ABB RAPID module: 0069C0E9

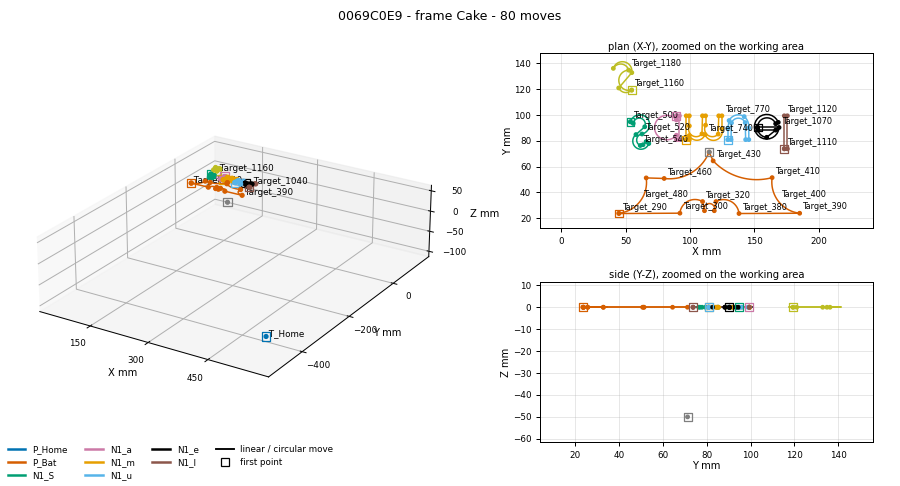
[picture p0: tool path of 0069C0E9 in frame Cake, 80 of 80 moves have a stored position in this frame; points joined in program order, loops and branches not executed]
MODULE Module1
    CONST robtarget T_Home:=[[572.610973065,-505,-40.400436373],[0,-0.000000007,0,1],[0,0,0,0],[9E+09,9E+09,9E+09,9E+09,9E+09,9E+09]];
    CONST robtarget Target_10:=[[44.887,23.575,0],[0.707106781,0,0,-0.707106781],[0,0,0,0],[9E+09,9E+09,9E+09,9E+09,9E+09,9E+09]];
    CONST robtarget Target_20:=[[91.921,23.575,0],[0.707106781,0,0,-0.707106781],[0,0,0,0],[9E+09,9E+09,9E+09,9E+09,9E+09,9E+09]];
    CONST robtarget Target_30:=[[93.942,29.137,0],[0.707106781,0,0,-0.707106781],[0,0,0,0],[9E+09,9E+09,9E+09,9E+09,9E+09,9E+09]];
    CONST robtarget Target_40:=[[97.861,32.778,0],[0.707106781,0,0,-0.707106781],[0,0,0,0],[9E+09,9E+09,9E+09,9E+09,9E+09,9E+09]];
    CONST robtarget Target_50:=[[101.269,33.587,0],[0.707106781,0,0,-0.707106781],[0,0,0,0],[9E+09,9E+09,9E+09,9E+09,9E+09,9E+09]];
    CONST robtarget Target_60:=[[104.374,34.284,0],[0.707106781,0,0,-0.707106781],[0,0,0,0],[9E+09,9E+09,9E+09,9E+09,9E+09,9E+09]];
    CONST robtarget Target_70:=[[107.601,34.604,0],[0.707106781,0,0,-0.707106781],[0,0,0,0],[9E+09,9E+09,9E+09,9E+09,9E+09,9E+09]];
    CONST robtarget Target_80:=[[109.794,32.852,0],[0.707106781,0,0,-0.707106781],[0,0,0,0],[9E+09,9E+09,9E+09,9E+09,9E+09,9E+09]];
    CONST robtarget Target_90:=[[111.194,25.675,0],[0.707106781,0,0,-0.707106781],[0,0,0,0],[9E+09,9E+09,9E+09,9E+09,9E+09,9E+09]];
    CONST robtarget Target_100:=[[112.426,30.409,0],[0.707106781,0,0,-0.707106781],[0,0,0,0],[9E+09,9E+09,9E+09,9E+09,9E+09,9E+09]];
    CONST robtarget Target_110:=[[115,30.175,0],[0.707106781,0,0,-0.707106781],[0,0,0,0],[9E+09,9E+09,9E+09,9E+09,9E+09,9E+09]];
    CONST robtarget Target_120:=[[117.574,30.409,0],[0.707106781,0,0,-0.707106781],[0,0,0,0],[9E+09,9E+09,9E+09,9E+09,9E+09,9E+09]];
    CONST robtarget Target_130:=[[118.806,25.675,0],[0.707106781,0,0,-0.707106781],[0,0,0,0],[9E+09,9E+09,9E+09,9E+09,9E+09,9E+09]];
    CONST robtarget Target_140:=[[120.206,32.852,0],[0.707106781,0,0,-0.707106781],[0,0,0,0],[9E+09,9E+09,9E+09,9E+09,9E+09,9E+09]];
    CONST robtarget Target_150:=[[122.399,34.604,0],[0.707106781,0,0,-0.707106781],[0,0,0,0],[9E+09,9E+09,9E+09,9E+09,9E+09,9E+09]];
    CONST robtarget Target_160:=[[125.626,34.284,0],[0.707106781,0,0,-0.707106781],[0,0,0,0],[9E+09,9E+09,9E+09,9E+09,9E+09,9E+09]];
    CONST robtarget Target_170:=[[128.731,33.587,0],[0.707106781,0,0,-0.707106781],[0,0,0,0],[9E+09,9E+09,9E+09,9E+09,9E+09,9E+09]];
    CONST robtarget Target_180:=[[132.139,32.778,0],[0.707106781,0,0,-0.707106781],[0,0,0,0],[9E+09,9E+09,9E+09,9E+09,9E+09,9E+09]];
    CONST robtarget Target_190:=[[136.058,29.137,0],[0.707106781,0,0,-0.707106781],[0,0,0,0],[9E+09,9E+09,9E+09,9E+09,9E+09,9E+09]];
    CONST robtarget Target_200:=[[137.882,23.65,0],[0.707106781,0,0,-0.707106781],[0,0,0,0],[9E+09,9E+09,9E+09,9E+09,9E+09,9E+09]];
    CONST robtarget Target_210:=[[185.214,23.669,0],[0.707106781,0,0,-0.707106781],[0,0,0,0],[9E+09,9E+09,9E+09,9E+09,9E+09,9E+09]];
    CONST robtarget Target_220:=[[168.341,33.479,0],[0.707106781,0,0,-0.707106781],[0,0,0,0],[9E+09,9E+09,9E+09,9E+09,9E+09,9E+09]];
    CONST robtarget Target_230:=[[163.916,51.359,0],[0.707106781,0,0,-0.707106781],[0,0,0,0],[9E+09,9E+09,9E+09,9E+09,9E+09,9E+09]];
    CONST robtarget Target_240:=[[135.263,52.898,0],[0.707106781,0,0,-0.707106781],[0,0,0,0],[9E+09,9E+09,9E+09,9E+09,9E+09,9E+09]];
    CONST robtarget Target_250:=[[114.922,71.263,0],[0.707106781,0,0,-0.707106781],[0,0,0,0],[9E+09,9E+09,9E+09,9E+09,9E+09,9E+09]];
    CONST robtarget Target_260:=[[94.738,52.898,0],[0.707106781,0,0,-0.707106781],[0,0,0,0],[9E+09,9E+09,9E+09,9E+09,9E+09,9E+09]];
    CONST robtarget Target_270:=[[66.084,51.359,0],[0.707106781,0,0,-0.707106781],[0,0,0,0],[9E+09,9E+09,9E+09,9E+09,9E+09,9E+09]];
    CONST robtarget Target_280:=[[61.659,33.479,0],[0.707106781,0,0,-0.707106781],[0,0,0,0],[9E+09,9E+09,9E+09,9E+09,9E+09,9E+09]];
    CONST robtarget Target_290:=[[44.887375283,23.575,0],[0.707106781,0,0,-0.707106781],[0,0,0,0],[9E+09,9E+09,9E+09,9E+09,9E+09,9E+09]];
    CONST robtarget Target_300:=[[92.217626762,23.834877014,0],[0.5,0,0,-0.866025404],[-1,0,-1,0],[9E+09,9E+09,9E+09,9E+09,9E+09,9E+09]];
    CONST robtarget Target_400:=[[168.340891695,33.478608179,0],[0.5,0,0,-0.866025404],[-1,0,-1,0],[9E+09,9E+09,9E+09,9E+09,9E+09,9E+09]];
    CONST robtarget Target_430:=[[118.021503486,64.425747652,0],[0.5,0,0,-0.866025404],[0,0,0,0],[9E+09,9E+09,9E+09,9E+09,9E+09,9E+09]];
    CONST robtarget Target_310:=[[97.860623741,32.777873993,0],[0.5,0,0,-0.866025404],[-1,0,-1,0],[9E+09,9E+09,9E+09,9E+09,9E+09,9E+09]];
    CONST robtarget Target_480:=[[61.659109682,33.478608179,0],[0.5,0,0,-0.866025404],[-1,0,-1,0],[9E+09,9E+09,9E+09,9E+09,9E+09,9E+09]];
    CONST robtarget Target_420:=[[135.262514114,52.897562122,0],[0.5,0,0,-0.866025404],[-1,0,-1,0],[9E+09,9E+09,9E+09,9E+09,9E+09,9E+09]];
    CONST robtarget Target_460:=[[79.985840188,50.770867258,0],[0.5,0,0,-0.866025404],[0,0,0,0],[9E+09,9E+09,9E+09,9E+09,9E+09,9E+09]];
    CONST robtarget Target_330:=[[111.283377266,25.744747734,0],[0.5,0,0,-0.866025404],[-1,0,-1,0],[9E+09,9E+09,9E+09,9E+09,9E+09,9E+09]];
    CONST robtarget Target_380:=[[138.079373741,23.575,0],[0.5,0,0,-0.866025404],[0,0,0,0],[9E+09,9E+09,9E+09,9E+09,9E+09,9E+09]];
    CONST robtarget Target_340:=[[112.525,30.426625252,0],[0.5,0,0,-0.866025404],[-1,0,-1,0],[9E+09,9E+09,9E+09,9E+09,9E+09,9E+09]];
    CONST robtarget Target_490:=[[44.854375315,23.789501762,0],[0.707106781,0,0,-0.707106781],[0,0,0,0],[9E+09,9E+09,9E+09,9E+09,9E+09,9E+09]];
    CONST robtarget Target_360:=[[120.205747986,32.852127266,0],[0.5,0,0,-0.866025404],[-1,0,-1,0],[9E+09,9E+09,9E+09,9E+09,9E+09,9E+09]];
    CONST robtarget Target_350:=[[118.898123741,25.740625,0],[0.5,0,0,-0.866025404],[0,0,0,0],[9E+09,9E+09,9E+09,9E+09,9E+09,9E+09]];
    CONST robtarget Target_370:=[[132.139376259,32.777873993,0],[0.5,0,0,-0.866025404],[-1,0,-1,0],[9E+09,9E+09,9E+09,9E+09,9E+09,9E+09]];
    CONST robtarget Target_410:=[[163.773995972,51.414627266,0],[0.5,0,0,-0.866025404],[0,0,0,0],[9E+09,9E+09,9E+09,9E+09,9E+09,9E+09]];
    CONST robtarget Target_470:=[[66.061000252,51.208377266,0],[0.5,0,0,-0.866025404],[-1,0,-1,0],[9E+09,9E+09,9E+09,9E+09,9E+09,9E+09]];
    CONST robtarget Target_320:=[[109.794252014,32.852127266,0],[0.5,0,0,-0.866025404],[0,0,0,0],[9E+09,9E+09,9E+09,9E+09,9E+09,9E+09]];
    CONST robtarget Target_440:=[[114.884500504,71.210504532,0],[0.5,0,0,-0.866025404],[-1,0,-1,0],[9E+09,9E+09,9E+09,9E+09,9E+09,9E+09]];
    CONST robtarget Target_450:=[[101.522546531,55.448907324,0],[0.5,0,0,-0.866025404],[-1,0,-1,0],[9E+09,9E+09,9E+09,9E+09,9E+09,9E+09]];
    CONST robtarget Target_390:=[[185.145619965,23.789501762,0],[0.5,0,0,-0.866025404],[-1,0,-1,0],[9E+09,9E+09,9E+09,9E+09,9E+09,9E+09]];
    CONST robtarget Target_500:=[[53.851116523,94.745073318,0],[0.707106781,0,0,-0.707106781],[0,0,0,0],[9E+09,9E+09,9E+09,9E+09,9E+09,9E+09]];
    CONST robtarget Target_510:=[[66.419099197,98.025150299,0],[0.707106781,0,0,-0.707106781],[-1,-1,0,0],[9E+09,9E+09,9E+09,9E+09,9E+09,9E+09]];
    CONST robtarget Target_520:=[[62.824605331,85.278720856,0],[0.707106781,0,0,-0.707106781],[0,0,0,0],[9E+09,9E+09,9E+09,9E+09,9E+09,9E+09]];
    CONST robtarget Target_530:=[[58.834970817,81.913661957,0],[0.707106781,0,0,-0.707106781],[-1,-1,0,0],[9E+09,9E+09,9E+09,9E+09,9E+09,9E+09]];
    CONST robtarget Target_540:=[[61.44799076,76.356220245,0],[0.707106781,0,0,-0.707106781],[0,0,0,0],[9E+09,9E+09,9E+09,9E+09,9E+09,9E+09]];
    CONST robtarget Target_550:=[[63.614881858,76.951055527,0],[0.707106781,0,0,-0.707106781],[-1,-1,0,0],[9E+09,9E+09,9E+09,9E+09,9E+09,9E+09]];
    CONST robtarget Target_560:=[[66.01970993,79.415369034,0],[0.707106781,0,0,-0.707106781],[-1,-1,0,0],[9E+09,9E+09,9E+09,9E+09,9E+09,9E+09]];
    CONST robtarget Target_570:=[[68.059137687,77.868800163,0],[0.707106781,0,0,-0.707106781],[-1,-1,0,0],[9E+09,9E+09,9E+09,9E+09,9E+09,9E+09]];
    CONST robtarget Target_580:=[[58.414338455,74.546232224,0],[0.707106781,0,0,-0.707106781],[-1,-1,0,0],[9E+09,9E+09,9E+09,9E+09,9E+09,9E+09]];
    CONST robtarget Target_590:=[[58.112676963,84.841098785,0],[0.707106781,0,0,-0.707106781],[0,0,0,0],[9E+09,9E+09,9E+09,9E+09,9E+09,9E+09]];
    CONST robtarget Target_600:=[[64.932015762,90.887155533,0],[0.707106781,0,0,-0.707106781],[-1,-1,0,0],[9E+09,9E+09,9E+09,9E+09,9E+09,9E+09]];
    CONST robtarget Target_610:=[[61.159070358,97.600269318,0],[0.707106781,0,0,-0.707106781],[-1,-1,0,0],[9E+09,9E+09,9E+09,9E+09,9E+09,9E+09]];
    CONST robtarget Target_620:=[[55.97552143,93.470430374,0],[0.707106781,0,0,-0.707106781],[0,0,0,0],[9E+09,9E+09,9E+09,9E+09,9E+09,9E+09]];
    CONST robtarget Target_630:=[[89.456146583,99.401769638,0],[0.608761429,0,0,-0.79335334],[0,0,0,0],[9E+09,9E+09,9E+09,9E+09,9E+09,9E+09]];
    CONST robtarget Target_640:=[[91.801489219,99.401769638,0],[0.608761429,0,0,-0.79335334],[-1,0,-1,0],[9E+09,9E+09,9E+09,9E+09,9E+09,9E+09]];
    CONST robtarget Target_650:=[[91.801489219,80.910949707,0],[0.608761429,0,0,-0.79335334],[-1,0,-1,0],[9E+09,9E+09,9E+09,9E+09,9E+09,9E+09]];
    CONST robtarget Target_660:=[[89.456146583,80.910949707,0],[0.608761429,0,0,-0.79335334],[-1,0,-1,0],[9E+09,9E+09,9E+09,9E+09,9E+09,9E+09]];
    CONST robtarget Target_670:=[[89.456146583,84.309997559,0],[0.608761429,0,0,-0.79335334],[-1,0,-1,0],[9E+09,9E+09,9E+09,9E+09,9E+09,9E+09]];
    CONST robtarget Target_680:=[[72.545884475,90.105371475,0],[0.608761429,0,0,-0.79335334],[-1,0,-1,0],[9E+09,9E+09,9E+09,9E+09,9E+09,9E+09]];
    CONST robtarget Target_690:=[[89.456146583,96.223659515,0],[0.608761429,0,0,-0.79335334],[0,0,0,0],[9E+09,9E+09,9E+09,9E+09,9E+09,9E+09]];
    CONST robtarget Target_700:=[[97.138002738,80.910949707,0],[0.608761429,0,0,-0.793353341],[0,0,0,0],[9E+09,9E+09,9E+09,9E+09,9E+09,9E+09]];
    CONST robtarget Target_710:=[[99.51732479,80.910949707,0],[0.608761429,0,0,-0.793353341],[-1,0,-1,0],[9E+09,9E+09,9E+09,9E+09,9E+09,9E+09]];
    CONST robtarget Target_720:=[[99.51732479,84.106054306,0],[0.608761429,0,0,-0.793353341],[-1,0,-1,0],[9E+09,9E+09,9E+09,9E+09,9E+09,9E+09]];
    CONST robtarget Target_730:=[[105.863989219,80.435085297,0],[0.608761429,0,0,-0.793353341],[-1,0,-1,0],[9E+09,9E+09,9E+09,9E+09,9E+09,9E+09]];
    CONST robtarget Target_740:=[[111.716993675,84.870834351,0],[0.608761429,0,0,-0.793353341],[0,0,0,0],[9E+09,9E+09,9E+09,9E+09,9E+09,9E+09]];
    CONST robtarget Target_750:=[[121.89846836,81.403808594,0],[0.608761429,0,0,-0.793353341],[-1,0,-1,0],[9E+09,9E+09,9E+09,9E+09,9E+09,9E+09]];
    CONST robtarget Target_760:=[[124.789255485,89.306592941,0],[0.608761429,0,0,-0.793353341],[0,0,0,0],[9E+09,9E+09,9E+09,9E+09,9E+09,9E+09]];
    CONST robtarget Target_770:=[[124.789255485,99.401769638,0],[0.608761429,0,0,-0.793353341],[-1,0,-1,0],[9E+09,9E+09,9E+09,9E+09,9E+09,9E+09]];
    CONST robtarget Target_780:=[[122.35893093,99.401769638,0],[0.608761429,0,0,-0.793353341],[-1,0,-1,0],[9E+09,9E+09,9E+09,9E+09,9E+09,9E+09]];
    CONST robtarget Target_790:=[[121.935518607,85.219240189,0],[0.608761429,0,0,-0.793353341],[-1,0,-1,0],[9E+09,9E+09,9E+09,9E+09,9E+09,9E+09]];
    CONST robtarget Target_800:=[[114.880369529,83.766145706,0],[0.608761429,0,0,-0.793353341],[-1,0,-1,0],[9E+09,9E+09,9E+09,9E+09,9E+09,9E+09]];
    CONST robtarget Target_810:=[[112.127798423,92.161798477,0],[0.608761429,0,0,-0.793353341],[0,0,0,0],[9E+09,9E+09,9E+09,9E+09,9E+09,9E+09]];
    CONST robtarget Target_820:=[[112.127798423,99.401769638,0],[0.608761429,0,0,-0.793353341],[-1,0,-1,0],[9E+09,9E+09,9E+09,9E+09,9E+09,9E+09]];
    CONST robtarget Target_830:=[[109.748466834,99.401769638,0],[0.608761429,0,0,-0.793353341],[-1,0,-1,0],[9E+09,9E+09,9E+09,9E+09,9E+09,9E+09]];
    CONST robtarget Target_840:=[[109.332083091,85.389194489,0],[0.608761429,0,0,-0.793353341],[-1,0,-1,0],[9E+09,9E+09,9E+09,9E+09,9E+09,9E+09]];
    CONST robtarget Target_850:=[[102.330044135,83.740653992,0],[0.608761429,0,0,-0.793353341],[-1,0,-1,0],[9E+09,9E+09,9E+09,9E+09,9E+09,9E+09]];
    CONST robtarget Target_860:=[[99.51732479,91.566963196,0],[0.608761429,0,0,-0.793353341],[0,0,0,0],[9E+09,9E+09,9E+09,9E+09,9E+09,9E+09]];
    CONST robtarget Target_870:=[[99.51732479,99.401769638,0],[0.608761429,0,0,-0.793353341],[-1,0,-1,0],[9E+09,9E+09,9E+09,9E+09,9E+09,9E+09]];
    CONST robtarget Target_880:=[[97.138002738,99.401769638,0],[0.608761429,0,0,-0.793353341],[-1,0,-1,0],[9E+09,9E+09,9E+09,9E+09,9E+09,9E+09]];
    CONST robtarget Target_890:=[[129.496935233,80.910949707,0],[0.5,0,0,-0.866025404],[0,0,0,0],[9E+09,9E+09,9E+09,9E+09,9E+09,9E+09]];
    CONST robtarget Target_900:=[[131.876266822,80.910949707,0],[0.5,0,0,-0.866025404],[-1,0,-1,0],[9E+09,9E+09,9E+09,9E+09,9E+09,9E+09]];
    CONST robtarget Target_910:=[[132.216699943,93.895311356,0],[0.5,0,0,-0.866025404],[-1,0,-1,0],[9E+09,9E+09,9E+09,9E+09,9E+09,9E+09]];
    CONST robtarget Target_920:=[[137.595165595,97.566280365,0],[0.5,0,0,-0.866025404],[-1,0,-1,0],[9E+09,9E+09,9E+09,9E+09,9E+09,9E+09]];
    CONST robtarget Target_930:=[[142.88864933,94.082260132,0],[0.5,0,0,-0.866025404],[0,0,0,0],[9E+09,9E+09,9E+09,9E+09,9E+09,9E+09]];
    CONST robtarget Target_940:=[[143.246086463,80.910949707,0],[0.5,0,0,-0.866025404],[-1,0,-1,0],[9E+09,9E+09,9E+09,9E+09,9E+09,9E+09]];
    CONST robtarget Target_950:=[[145.676401481,80.910949707,0],[0.5,0,0,-0.866025404],[-1,0,-1,0],[9E+09,9E+09,9E+09,9E+09,9E+09,9E+09]];
    CONST robtarget Target_1000:=[[145.676,89.986,0],[0.5,0,0,-0.866025404],[-1,0,-1,0],[9E+09,9E+09,9E+09,9E+09,9E+09,9E+09]];
    CONST robtarget Target_960:=[[145.453346595,93.338718414,0],[0.5,0,0,-0.866025404],[-1,0,-1,0],[9E+09,9E+09,9E+09,9E+09,9E+09,9E+09]];
    CONST robtarget Target_970:=[[142.098911628,98.781442642,0],[0.5,0,0,-0.866025404],[-1,0,-1,0],[9E+09,9E+09,9E+09,9E+09,9E+09,9E+09]];
    CONST robtarget Target_980:=[[133.091429099,98.781442642,0],[0.5,0,0,-0.866025404],[-1,0,-1,0],[9E+09,9E+09,9E+09,9E+09,9E+09,9E+09]];
    CONST robtarget Target_1010:=[[130.389,95.722,0],[0.5,0,0,-0.866025404],[-1,0,-1,0],[9E+09,9E+09,9E+09,9E+09,9E+09,9E+09]];
    CONST robtarget Target_990:=[[129.496935233,89.816455841,0],[0.5,0,0,-0.866025404],[0,0,0,0],[9E+09,9E+09,9E+09,9E+09,9E+09,9E+09]];
    CONST robtarget Target_1020:=[[152.508495674,90.34330368,0],[0.5,0,0,-0.866025404],[0,0,0,0],[9E+09,9E+09,9E+09,9E+09,9E+09,9E+09]];
    CONST robtarget Target_1030:=[[156.792162284,97.170209885,0],[0.5,0,0,-0.866025404],[-1,0,-1,0],[9E+09,9E+09,9E+09,9E+09,9E+09,9E+09]];
    CONST robtarget Target_1040:=[[166.529577598,93.266487122,0],[0.5,0,0,-0.866025404],[0,0,0,0],[9E+09,9E+09,9E+09,9E+09,9E+09,9E+09]];
    CONST robtarget Target_1050:=[[168.535002097,94.320192337,0],[0.5,0,0,-0.866025404],[-1,0,-1,0],[9E+09,9E+09,9E+09,9E+09,9E+09,9E+09]];
    CONST robtarget Target_1060:=[[150.061176643,90.20734787,0],[0.5,0,0,-0.866025404],[-1,0,-1,0],[9E+09,9E+09,9E+09,9E+09,9E+09,9E+09]];
    CONST robtarget Target_1070:=[[169.146841392,90.34330368,0],[0.5,0,0,-0.866025404],[0,0,0,0],[9E+09,9E+09,9E+09,9E+09,9E+09,9E+09]];
    CONST robtarget Target_1020_2:=[[152.508495674,90.34330368,0],[0.5,0,0,-0.866025404],[0,0,0,0],[9E+09,9E+09,9E+09,9E+09,9E+09,9E+09]];
    CONST robtarget Target_1080:=[[152.746,88.287,0],[0.5,0,0,-0.866025404],[-1,0,-1,0],[9E+09,9E+09,9E+09,9E+09,9E+09,9E+09]];
    CONST robtarget Target_1090:=[[159.587,82.712,0],[0.5,0,0,-0.866025404],[-1,0,-1,0],[9E+09,9E+09,9E+09,9E+09,9E+09,9E+09]];
    CONST robtarget Target_1100:=[[166.53,88.287,0],[0.5,0,0,-0.866025404],[-1,0,-1,0],[9E+09,9E+09,9E+09,9E+09,9E+09,9E+09]];
    CONST robtarget Target_1110:=[[173.225706443,73.772945404,0],[0.5,0,0,-0.866025404],[0,0,0,0],[9E+09,9E+09,9E+09,9E+09,9E+09,9E+09]];
    CONST robtarget Target_1120:=[[173.225706443,99.401769638,0],[0.5,0,0,-0.866025404],[-1,0,-1,0],[9E+09,9E+09,9E+09,9E+09,9E+09,9E+09]];
    CONST robtarget Target_1130:=[[175.605028495,99.401769638,0],[0.5,0,0,-0.866025404],[-1,0,-1,0],[9E+09,9E+09,9E+09,9E+09,9E+09,9E+09]];
    CONST robtarget Target_1140:=[[175.605028495,73.772945404,0],[0.5,0,0,-0.866025404],[-1,0,-1,0],[9E+09,9E+09,9E+09,9E+09,9E+09,9E+09]];
    CONST robtarget Target_1150:=[[173.225706443,73.772945404,0],[0.5,0,0,-0.866025404],[-1,0,-1,0],[9E+09,9E+09,9E+09,9E+09,9E+09,9E+09]];
    CONST robtarget T_Local_Home:=[[115.079,71.263,-50],[0.707106781,0.000000005,-0.000000005,-0.707106781],[0,0,0,0],[9E+09,9E+09,9E+09,9E+09,9E+09,9E+09]];

    ! Variable para almacenar posición temporal
    VAR robtarget current_pos;
    CONST robtarget Target_1160:=[[54.76886116,119.337177277,0],[0.446392083,0,0,-0.894837476],[0,0,0,0],[9E+09,9E+09,9E+09,9E+09,9E+09,9E+09]];
    CONST robtarget Target_1170:=[[44.822400436,126.309480667,0],[0.36650971,0,0,-0.930414226],[0,0,0,0],[9E+09,9E+09,9E+09,9E+09,9E+09,9E+09]];
    CONST robtarget Target_1180:=[[52.491501197,134.819850922,0],[0.740357165,0,0,0.672213707],[0,0,0,0],[9E+09,9E+09,9E+09,9E+09,9E+09,9E+09]];
    CONST robtarget Target_1190:=[[49.088199958,138.922071457,0],[0.121523417,0,0,0.992588565],[0,0,0,0],[9E+09,9E+09,9E+09,9E+09,9E+09,9E+09]];
    CONST robtarget Target_1200:=[[40.560839996,136.2134552,0],[0.266933582,0,0,0.963714928],[0,0,0,0],[9E+09,9E+09,9E+09,9E+09,9E+09,9E+09]];
    CONST robtarget Target_1210:=[[45.935591087,141.1951828,0],[0.989624414,0,0,0.143678526],[0,0,0,0],[9E+09,9E+09,9E+09,9E+09,9E+09,9E+09]];
    CONST robtarget Target_1220:=[[54.89208065,132.886638641,0],[0.594295659,0,0,-0.804246648],[0,0,0,0],[9E+09,9E+09,9E+09,9E+09,9E+09,9E+09]];
    CONST robtarget Target_1230:=[[44.724677429,121.00271225,0],[0.687884928,0,0,-0.725819761],[0,0,0,0],[9E+09,9E+09,9E+09,9E+09,9E+09,9E+09]];
    CONST robtarget Target_1240:=[[48.157714233,117.824602127,0],[0.999420129,0,0,-0.034050051],[0,0,0,0],[9E+09,9E+09,9E+09,9E+09,9E+09,9E+09]];
    CONST robtarget Target_1250:=[[54.76886116,119.337177277,0],[0.94783967,0,0,-0.318747487],[0,0,0,0],[9E+09,9E+09,9E+09,9E+09,9E+09,9E+09]];

    PROC main()
        ! 1. Ir a Home
        P_Home;

        ! 2. Ir a Local Home
        P_Local_Home;

        ! 3. Ejecutar P_Bat y subir 50mm
        P_Bat;P_Local_Home;
        !current_pos := CRobT(\Tool:=Marker\WObj:=Cake);
        !current_pos.trans.z := current_pos.trans.z + 50;
        !MoveL current_pos, v100, z5, Marker\WObj:=Cake;

        ! 4. Ejecutar N1_S y subir 50mm
        N1_S;P_Local_Home;
        !current_pos := CRobT(\Tool:=Marker\WObj:=Cake);
        !current_pos.trans.z := current_pos.trans.z + 50;
        !MoveL current_pos, v100, z5, Marker\WObj:=Cake;

        ! 5. Ejecutar N1_a y subir 50mm
        N1_a;P_Local_Home;
        !current_pos := CRobT(\Tool:=Marker\WObj:=Cake);
        !current_pos.trans.z := current_pos.trans.z + 50;
        !MoveL current_pos, v100, z5, Marker\WObj:=Cake;

        ! 6. Ejecutar N1_m y subir 50mm
        N1_m;P_Local_Home;
        !current_pos := CRobT(\Tool:=Marker\WObj:=Cake);
        !current_pos.trans.z := current_pos.trans.z + 50;
        !MoveL current_pos, v300, z5, Marker\WObj:=Cake;

        ! 7. Ejecutar N1_u y subir 50mm
        N1_u;P_Local_Home;
        !current_pos := CRobT(\Tool:=Marker\WObj:=Cake);
        !current_pos.trans.z := current_pos.trans.z + 50;
        !MoveL current_pos, v300, z5, Marker\WObj:=Cake;

        ! 8. Ejecutar N1_e y subir 50mm
        N1_e;P_Local_Home;
        !current_pos := CRobT(\Tool:=Marker\WObj:=Cake);
        !current_pos.trans.z := current_pos.trans.z + 50;
        !MoveL current_pos, v100, z5, Marker\WObj:=Cake;

        ! 9. Ejecutar N1_l y subir 50mm
        N1_l;P_Local_Home;
        !current_pos := CRobT(\Tool:=Marker\WObj:=Cake);
        !current_pos.trans.z := current_pos.trans.z + 50;
        !MoveL current_pos, v100, z5, Marker\WObj:=Cake;

        ! Opcional: Volver a Home al finalizar
        P_Local_Home;P_Home;

    ENDPROC
    PROC P_Home()
        MoveL T_Home,v300,z50,Marker\WObj:=Cake;
    ENDPROC
    PROC P_Bat()
        MoveL Target_290,v150,z5,Marker\WObj:=Cake;
        MoveL Target_300,v150,z5,Marker\WObj:=Cake;
        MoveC Target_310,Target_320,v150,z5,Marker\WObj:=Cake;
        MoveL Target_330,v150,z5,Marker\WObj:=Cake;
        MoveC Target_340,Target_350,v150,z5,Marker\WObj:=Cake;
        MoveL Target_360,v150,z5,Marker\WObj:=Cake;
        MoveC Target_370,Target_380,v150,z5,Marker\WObj:=Cake;
        MoveL Target_390,v150,z5,Marker\WObj:=Cake;
        MoveC Target_400,Target_410,v150,z5,Marker\WObj:=Cake;
        MoveC Target_420,Target_430,v150,z5,Marker\WObj:=Cake;
        MoveL Target_440,v150,z5,Marker\WObj:=Cake;
        MoveC Target_450,Target_460,v150,z5,Marker\WObj:=Cake;
        MoveL Target_470,v150,z5,Marker\WObj:=Cake;
        MoveC Target_480,Target_490,v150,z5,Marker\WObj:=Cake;
    ENDPROC
    PROC N1_S()
        MoveL Target_500,v1000,z100,Marker\WObj:=Cake;
        MoveC Target_510,Target_520,v1000,z100,Marker\WObj:=Cake;
        MoveC Target_530,Target_540,v1000,z100,Marker\WObj:=Cake;
        MoveL Target_550,v1000,z100,Marker\WObj:=Cake;
        MoveL Target_560,v1000,z100,Marker\WObj:=Cake;
        MoveL Target_570,v1000,z100,Marker\WObj:=Cake;
        MoveC Target_580,Target_590,v1000,z100,Marker\WObj:=Cake;
        MoveL Target_600,v1000,z100,Marker\WObj:=Cake;
        MoveC Target_610,Target_620,v1000,z100,Marker\WObj:=Cake;
        MoveL Target_500,v1000,z100,Marker\WObj:=Cake;
    ENDPROC
    PROC N1_a()
        MoveL Target_630,v150,z5,Marker\WObj:=Cake;
        MoveL Target_640,v150,z5,Marker\WObj:=Cake;
        MoveL Target_650,v150,z5,Marker\WObj:=Cake;
        MoveL Target_660,v150,z5,Marker\WObj:=Cake;
        MoveL Target_670,v150,z5,Marker\WObj:=Cake;
        MoveC Target_680,Target_690,v150,z5,Marker\WObj:=Cake;
        MoveL Target_630,v150,z5,Marker\WObj:=Cake;
    ENDPROC
    PROC N1_m()
        MoveL Target_700,v150,z5,Marker\WObj:=Cake;
        MoveL Target_710,v150,z5,Marker\WObj:=Cake;
        MoveL Target_720,v150,z5,Marker\WObj:=Cake;
        MoveC Target_730,Target_740,v150,z5,Marker\WObj:=Cake;
        MoveC Target_750,Target_760,v150,z5,Marker\WObj:=Cake;
        MoveL Target_770,v150,z5,Marker\WObj:=Cake;
        MoveL Target_780,v150,z5,Marker\WObj:=Cake;
        MoveL Target_790,v150,z5,Marker\WObj:=Cake;
        MoveC Target_800,Target_810,v150,z5,Marker\WObj:=Cake;
        MoveL Target_820,v150,z5,Marker\WObj:=Cake;
        MoveL Target_830,v150,z5,Marker\WObj:=Cake;
        MoveL Target_840,v150,z5,Marker\WObj:=Cake;
        MoveC Target_850,Target_860,v150,z5,Marker\WObj:=Cake;
        MoveL Target_870,v150,z5,Marker\WObj:=Cake;
        MoveL Target_880,v150,z5,Marker\WObj:=Cake;
        MoveL Target_700,v150,z5,Marker\WObj:=Cake;
    ENDPROC
    PROC N1_u()
        MoveL Target_890,v150,z5,Marker\WObj:=Cake;
        MoveL Target_900,v150,z5,Marker\WObj:=Cake;
        MoveL Target_910,v150,z5,Marker\WObj:=Cake;
        MoveC Target_920,Target_930,v150,z5,Marker\WObj:=Cake;
        MoveL Target_940,v150,z5,Marker\WObj:=Cake;
        MoveL Target_950,v150,z5,Marker\WObj:=Cake;
        MoveL Target_1000,v150,z5,Marker\WObj:=Cake;
        MoveC Target_960,Target_970,v150,z5,Marker\WObj:=Cake;
        MoveC Target_980,Target_1010,v150,z5,Marker\WObj:=Cake;
        MoveL Target_990,v150,z5,Marker\WObj:=Cake;
        MoveL Target_890,v150,z5,Marker\WObj:=Cake;
    ENDPROC
    PROC N1_e()
        MoveL Target_1020,v150,z5,Marker\WObj:=Cake;
        MoveC Target_1030,Target_1040,v150,z5,Marker\WObj:=Cake;
        MoveL Target_1050,v150,z5,Marker\WObj:=Cake;
        MoveC Target_1060,Target_1070,v150,z5,Marker\WObj:=Cake;
        MoveL Target_1020,v150,z5,Marker\WObj:=Cake;
        MoveL Target_1020_2,v150,z5,Marker\WObj:=Cake;
        MoveC Target_1080,Target_1090,v150,z5,Marker\WObj:=Cake;
        MoveC Target_1090,Target_1100,v150,z5,Marker\WObj:=Cake;
        MoveL Target_1080,v150,z5,Marker\WObj:=Cake;
    ENDPROC
    PROC N1_l()
        MoveL Target_1110,v150,z5,Marker\WObj:=Cake;
        MoveL Target_1120,v150,z5,Marker\WObj:=Cake;
        MoveL Target_1130,v150,z5,Marker\WObj:=Cake;
        MoveL Target_1140,v150,z5,Marker\WObj:=Cake;
        MoveL Target_1150,v150,z5,Marker\WObj:=Cake;
    ENDPROC
    PROC P_Local_Home()
        MoveL T_Local_Home,v300,z5,Marker\WObj:=Cake;
    ENDPROC
    PROC Path_10()
        MoveL Target_1160,v1000,z100,Marker\WObj:=Cake;
        MoveC Target_1170,Target_1180,v1000,z100,Marker\WObj:=Cake;
        MoveC Target_1190,Target_1200,v1000,z100,Marker\WObj:=Cake;
        MoveC Target_1210,Target_1220,v1000,z100,Marker\WObj:=Cake;
        MoveL Target_1230,v1000,z100,Marker\WObj:=Cake;
        MoveC Target_1240,Target_1250,v1000,z100,Marker\WObj:=Cake;
    ENDPROC
    PROC Path_20()

    ENDPROC
ENDMODULE
